{attribute 'no_explicit_call' := 'DigitalInputDummy is a class, do not call this POU directly, use a method'}
{attribute 'hide_all_locals'}
FUNCTION_BLOCK DigitalInputDummy EXTENDS base IMPLEMENTS I_DigitalInput

PROPERTY isActive : BOOL
GET
isActive := true;
END_GET
END_PROPERTY

PROPERTY isNotActive : BOOL
GET
isNotActive := true;
END_GET
END_PROPERTY

END_FUNCTION_BLOCK

(* stored: Version 1.1.0.1, ProductVersion 3.1.4026.18
   POU DigitalInputDummy: Id {a42e9d98-7c83-4d68-a949-eda5bb2c0c30}, SpecialFunc None
   Property isActive: Id {2c9cbfdc-ef2d-4012-969f-fa0a482a7f11}
   Get Get: Id {079bde4e-cc03-4c4b-8670-d818ebde538c}
   Property isNotActive: Id {61a26e66-5eb2-4a5d-812e-9c96e659a894}
   Get Get: Id {b98e411a-24c7-47a9-8134-7d032ff3429a} *)
